(* CoDeSys 2.3.9.50 project: 9A.pr6 *)
(* Libraries: STANDARD.LB6 5.6.98 12:03:02 *)

(* POU MAIN, LD *)
PROGRAM MAIN
VAR
	Start AT %IX0.0: BOOL;
	value: INT := 23;
	a AT %QX0.0: BOOL;
	Heater1 AT %QX0.1: BOOL;
	T1: TOF;
	b AT %QX0.3: BOOL;
	Heater2 AT %QX0.4: BOOL;
	T2: TOF;
	c AT %QX0.5: BOOL;
	Heater3 AT %QX0.6: BOOL;
	T3: TOF;
	d AT %IX0.7: BOOL;
	Increase_Pressure AT %IX2.0: BOOL;
	Current_Pressure: INT := 0;
	Final: INT;
	Decrease_Pressure AT %IX2.1: BOOL;
	ON AT %QX2.0: BOOL;
	NO_more AT %QX2.1: BOOL;
	NO_less AT %QX2.2: BOOL;
END_VAR
VAR (* helpers for the ST form of the networks *)
	_p1 : BOOL;
	_p2 : BOOL;
	_p3 : BOOL;
END_VAR
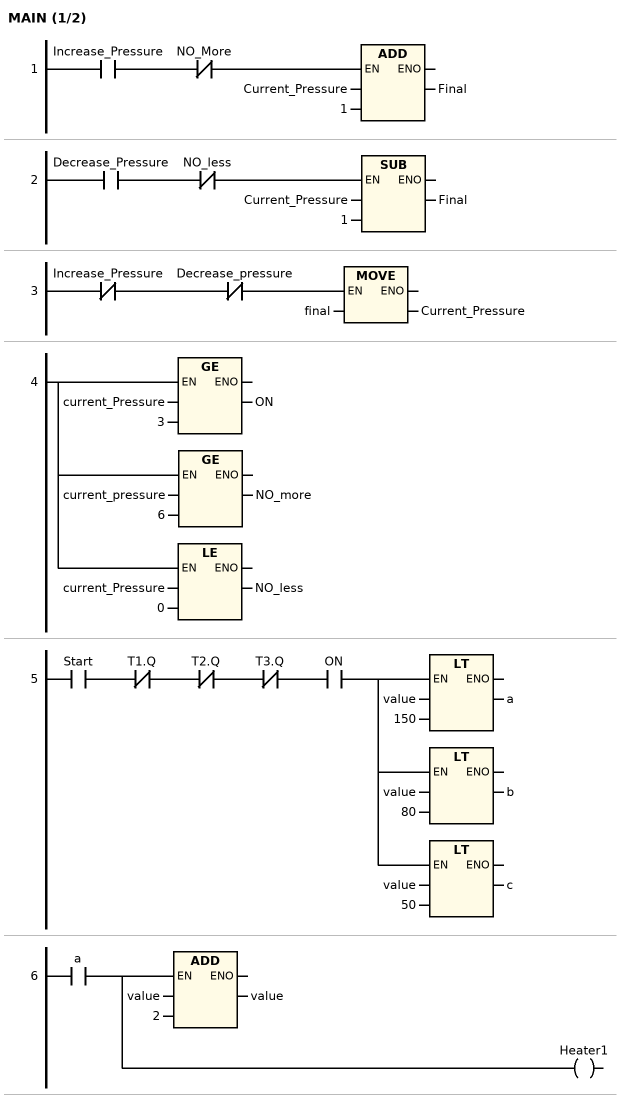
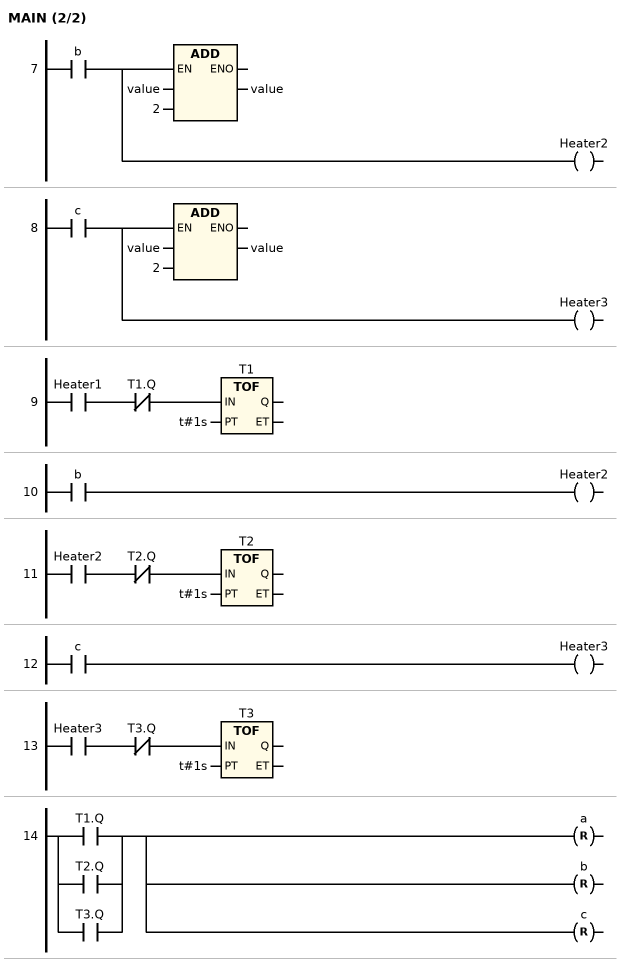
_LD_ (* Ladder Diagram *)
NETWORK 1
	[Increase_Pressure] - [/NO_More]
		EN --- ADD(Current_Pressure, 1) => Final
NETWORK 2
	[Decrease_Pressure] - [/NO_less]
		EN --- SUB(Current_Pressure, 1) => Final
NETWORK 3
	[/Increase_Pressure] - [/Decrease_pressure]
		EN --- MOVE(final) => Current_Pressure
NETWORK 4
	*
		EN --- GE(current_Pressure, 3) => ON
		EN --- GE(current_pressure, 6) => NO_more
		EN --- LE(current_Pressure, 0) => NO_less
NETWORK 5
	[Start] - [/T1.Q] - [/T2.Q] - [/T3.Q] - [ON]
		EN --- LT(value, 150) => a
		EN --- LT(value, 80) => b
		EN --- LT(value, 50) => c
NETWORK 6
	[a] --- (Heater1)
		EN --- ADD(value, 2) => value
NETWORK 7
	[b] --- (Heater2)
		EN --- ADD(value, 2) => value
NETWORK 8
	[c] --- (Heater3)
		EN --- ADD(value, 2) => value
NETWORK 9
	[Heater1] - [/T1.Q] - T1:TOF(IN: *, PT: t#1s)
NETWORK 10
	[b] --- (Heater2)
NETWORK 11
	[Heater2] - [/T2.Q] - T2:TOF(IN: *, PT: t#1s)
NETWORK 12
	[c] --- (Heater3)
NETWORK 13
	[Heater3] - [/T3.Q] - T3:TOF(IN: *, PT: t#1s)
NETWORK 14
	{ [T1.Q] | [T2.Q] | [T3.Q] } --- (R a) (R b) (R c)
_END_LD_
(* the same logic as Structured Text *)
(* Network 1 *)
IF Increase_Pressure AND NOT NO_More THEN
	Final := Current_Pressure + 1;
END_IF;
(* Network 2 *)
IF Decrease_Pressure AND NOT NO_less THEN
	Final := Current_Pressure - 1;
END_IF;
(* Network 3 *)
IF NOT Increase_Pressure AND NOT Decrease_pressure THEN
	Current_Pressure := final;
END_IF;
(* Network 4 *)
ON := current_Pressure >= 3;
NO_more := current_pressure >= 6;
NO_less := current_Pressure <= 0;
(* Network 5 *)
IF Start AND NOT T1.Q AND NOT T2.Q AND NOT T3.Q AND ON THEN
	a := value < 150;
	b := value < 80;
	c := value < 50;
END_IF;
(* Network 6 *)
_p1 := a;
IF _p1 THEN
	value := value + 2;
END_IF;
Heater1 := _p1;
(* Network 7 *)
_p2 := b;
IF _p2 THEN
	value := value + 2;
END_IF;
Heater2 := _p2;
(* Network 8 *)
_p3 := c;
IF _p3 THEN
	value := value + 2;
END_IF;
Heater3 := _p3;
(* Network 9 *)
T1(IN := Heater1 AND NOT T1.Q, PT := t#1s);
(* Network 10 *)
Heater2 := b;
(* Network 11 *)
T2(IN := Heater2 AND NOT T2.Q, PT := t#1s);
(* Network 12 *)
Heater3 := c;
(* Network 13 *)
T3(IN := Heater3 AND NOT T3.Q, PT := t#1s);
(* Network 14 *)
IF T1.Q OR T2.Q OR T3.Q THEN a := FALSE; b := FALSE; c := FALSE; END_IF;
END_PROGRAM
